// TIA Portal V17 export
// export: Created 2023-12-22T15:28:36.4496848Z, ExportSetting WithDefaults, DisplayName Totally Integrated Automation Portal, DisplayVersion V17, DisplayName TIA Portal Openness, DisplayVersion V17, DisplayName TIA Portal Version Control Interface, DisplayVersion V17, DisplayName STEP 7 Professional, DisplayVersion V17, DisplayName STEP 7 Safety, DisplayVersion V17, DisplayName WinCC Advanced, DisplayVersion V17
DATA_BLOCK "AO_example_DB"   // DB400
VERSION : 0.1
// stored: AutoNumber false, DBAccessibleFromOPCUA true, InstanceOfName AO_ex, InstanceOfType FB
"AO_ex"
   // VAR_INPUT
   //    SP_A : Real;
   //    All_Block : Bool;
   // END_VAR
   // VAR_IN_OUT
   //    Signal : Int;
   // END_VAR
   // VAR RETAIN
   //    CMD : "CMD";
   //    Mode : Int;
   //    Status : Int;
   //    Use : Struct
   //       Indirect { S7_SetPoint := 'True'} : Bool;
   //    END_STRUCT;
   //    VmA : Real;
   //    SP_M : Real;
   //    Converter { S7_SetPoint := 'True'} : "Converter";
   //    Events : Word;
   //    pos : Array[0..15] of Bool;
   //    Output_Type { S7_SetPoint := 'True'} : Int;
   //    CodeID { S7_SetPoint := 'True'} : Int;
   //    "Type" { S7_SetPoint := 'True'} : Int;
   //    ADDR { S7_SetPoint := 'True'} : Int;
   //    Slow { S7_SetPoint := 'True'} : "Slow";
   //    Time_DTL { S7_SetPoint := 'True'} : DTL;
   // END_VAR
BEGIN
END_DATA_BLOCK
